% RSLogix 500 project ONE BUTTON BITS_BAK017.RSS, saved by version 10.00.00.00 %
PROJECT "MWL"    % processor: Bul.1763 MicroLogix 1100 Series B %

PROGRAM FILES
  LAD 2 "MAIN"  4 rungs

DATA FILES
  O0 OUTPUT  4 elements
  I1 INPUT  6 elements
  S2 STATUS  66 elements
  B3 BINARY  2 elements
  T4 TIMER  1 elements
  C5 COUNTER  1 elements
  R6 CONTROL  1 elements
  N7 INTEGER  1 elements
  F8 FLOAT  1 elements

LADDER 2 "MAIN"
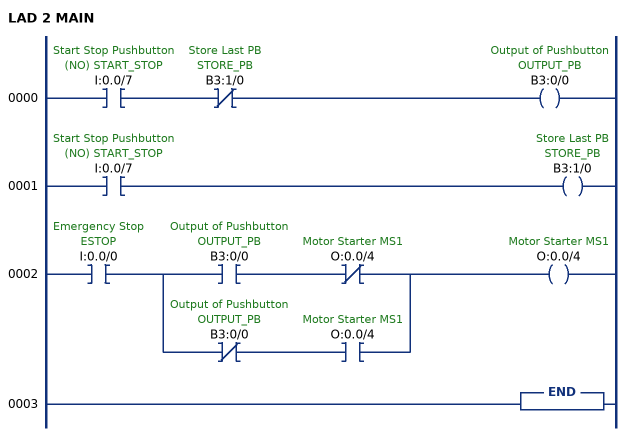
% Rung: 0 %
SOR XIC I:0.0/7 XIO B3:1/0 OTE B3:0/0 EOR
%   I:0.0/7  START_STOP  "Start Stop Pushbutton (NO)" %
%   B3:1/0  STORE_PB  "Store Last PB" %
%   B3:0/0  OUTPUT_PB  "Output of Pushbutton" %
% Rung: 1 %
SOR XIC I:0.0/7 OTE B3:1/0 EOR
%   I:0.0/7  START_STOP  "Start Stop Pushbutton (NO)" %
%   B3:1/0  STORE_PB  "Store Last PB" %
% Rung: 2 %
SOR XIC I:0.0/0 BST XIC B3:0/0 XIO O:0.0/4 NXB XIO B3:0/0 XIC O:0.0/4 BND OTE O:0.0/4 EOR
%   I:0.0/0  ESTOP  "Emergency Stop" %
%   B3:0/0  OUTPUT_PB  "Output of Pushbutton" %
%   O:0.0/4  MS1  "Motor Starter" %
% Rung: 3 %
SOR END EOR

OTHER DOCUMENTED ADDRESSES
  U:3  ONE_PB
